(* IEC 61131-3 sources: sps_maggio25/src/Program, 5 files *)

(* ---- CustomTypes.st ---- *)
NAMESPACE ProgramCustomTypes

    TYPE
        TankState : (Stopped, Filling, Emptying):= Stopped;
    END_TYPE

END_NAMESPACE

(* ---- ITank.st ---- *)
INTERFACE ITank
    METHOD OpenInletValve
    END_METHOD

    METHOD OpenOutletValve
    END_METHOD

    METHOD CloseInletValve
    END_METHOD

    METHOD CloseOutletValve
    END_METHOD

    METHOD Fill
    END_METHOD

    METHOD Close
    END_METHOD

    METHOD Flush
    END_METHOD

END_INTERFACE

(* ---- Tank.st ---- *)
USING Libreria.Moduli;

NAMESPACE ProgramModuli

    CLASS Tank IMPLEMENTS ITank

        VAR PUBLIC
            inletValve : ClassValve;
            outletValve : ClassValve;
        END_VAR

        METHOD PUBLIC OpenInletValve
            inletValve.Open();
        END_METHOD

        METHOD PUBLIC OpenOutletValve
            outletValve.Open();
        END_METHOD

        METHOD PUBLIC CloseInletValve
            inletValve.Close();
        END_METHOD

        METHOD PUBLIC CloseOutletValve
            outletValve.Close();
        END_METHOD

        METHOD PUBLIC Fill
            THIS.OpenInletValve();
            THIS.CloseOutletValve();
        END_METHOD

        METHOD PUBLIC Close
            THIS.CloseInletValve();
            THIS.CloseOutletValve();
        END_METHOD

        METHOD PUBLIC Flush
            THIS.OpenInletValve();
            THIS.OpenOutletValve();
        END_METHOD

    END_CLASS

END_NAMESPACE

(* ---- TankRegulatorDelayed.st ---- *)
USING Libreria.Moduli;
USING System.Timer;
USING ProgramModuli;
USING ProgramCustomTypes;

NAMESPACE directloading.ModuliOOP
    FUNCTION_BLOCK TankRegulatorDelayed
        VAR_INPUT
            enable: BOOL;
            tank : REF_TO Tank;
        END_VAR
        VAR
            stateTankMachine : TankState := TankState#Stopped;
            timer : OnDelay;
        END_VAR

        IF NOT enable THEN
            stateTankMachine := TankState#Stopped;
        END_IF;

        CASE stateTankMachine OF

            TankState#Stopped:
                tank^.Close();
                timer(signal:=false, duration:=LT#0s);
                IF enable THEN
                    stateTankMachine:= TankState#Filling;
                END_IF;

            TankState#Filling:
                timer(signal:=true, duration:=LT#10s);
                tank^.Fill();
                IF timer.output THEN
                    stateTankMachine:= TankState#Emptying;
                    timer(signal:=false, duration:=LT#0s);
                END_IF;

            TankState#Emptying:
                timer(signal:=true, duration:=LT#10s);
                tank^.Flush();
                IF timer.output THEN
                    stateTankMachine:= TankState#Filling;
                    timer(signal:=false, duration:=LT#0s);
                END_IF;
        END_CASE;
    END_FUNCTION_BLOCK
END_NAMESPACE

(* ---- MainProgram.st ---- *)
USING System.Timer;
USING ProgramModuli;
USING ProgramCustomTypes;

PROGRAM MainProgram
    VAR_EXTERNAL
        //use lamp to import global variables from Configuration
        enable: BOOL;
        tank : Tank;
        ctrlInletOpen : BOOL;
        ctrlOutletOpen : BOOL;
    END_VAR

    VAR
        stateTankMachine : TankState := TankState#Stopped;
        timer : OnDelay;
    END_VAR

    VAR CONSTANT
        speedAxisDB  : UINT := UINT#1;
    END_VAR

    // state machine
    IF NOT enable THEN
        stateTankMachine := TankState#Stopped;
    END_IF;

    CASE stateTankMachine OF

        TankState#Stopped:
            tank.Close();
            timer(signal:=false, duration:=LT#0s);
            IF enable THEN
                stateTankMachine:= TankState#Filling;
            END_IF;

        TankState#Filling:
            timer(signal:=true, duration:=LT#10s);
            tank.Fill();
            IF timer.output THEN
                stateTankMachine:= TankState#Emptying;
                timer(signal:=false, duration:=LT#0s);
            END_IF;

        TankState#Emptying:
            timer(signal:=true, duration:=LT#10s);
            tank.Flush();
            IF timer.output THEN
                stateTankMachine:= TankState#Filling;
                timer(signal:=false, duration:=LT#0s);
            END_IF;
    END_CASE;

    // connection to the Tanks --> we need to pass them to FB inputs!
    ctrlInletOpen:=tank.inletValve.ctrlOpen;
    ctrlOutletOpen:=tank.outletValve.ctrlOpen;

END_PROGRAM
